(* IEC 61131-3 sources: ecmc_strucpp_app_example/st, 7 files *)

(* ---- el7041_velocity.st ---- *)
PROGRAM EL7041_VELOCITY
VAR
  actual_position    AT %IW0 : INT;   // @ecmc ec0.s14.positionActual01
  drive_control      AT %QW0 : WORD;  // @ecmc ec0.s14.driveControl01
  velocity_setpoint  AT %QW2 : INT;   // @ecmc ec0.s14.velocitySetpoint01
END_VAR

drive_control := 16#0001;
velocity_setpoint := 1000;
END_PROGRAM

(* ---- machine.st ---- *)
PROGRAM MACHINE
VAR
  start_button   AT %IX0.0 : BOOL;  // @ecmc ec0.s2.mm.inputDataArray01
  stop_button    AT %IX0.1 : BOOL;  // @ecmc ec0.s2.mm.inputDataArray01
  enable_output  AT %QX0.0 : BOOL;  // @ecmc ec0.s2.mm.outputDataArray01
  target_word    AT %QW2   : INT;   // @ecmc ec0.s2.mm.outputDataArray01
  counter        AT %MW0   : INT;
END_VAR

IF stop_button THEN
  enable_output := FALSE;
ELSIF start_button THEN
  enable_output := TRUE;
END_IF;

IF enable_output THEN
  counter := counter + 1;
  target_word := counter;
ELSE
  target_word := 0;
END_IF;
END_PROGRAM

(* ---- mc_power_move_absolute_lib.st ---- *)
PROGRAM MC_POWER_MOVE_ABSOLUTE_LIB
VAR
  axis        : ECMC_AXIS_REF;
  power       : MC_Power;
  moveAbs     : MC_MoveAbsolute;
  readPos     : MC_ReadActualPosition;

  enableCmd   AT %IX0.0 : BOOL;
  executeCmd  AT %IX0.1 : BOOL;

  targetPos   AT %IL8  : LREAL;
  velocity    AT %IL16 : LREAL;
  accel       AT %IL24 : LREAL;
  decel       AT %IL32 : LREAL;

  powerStatus AT %QX0.0 : BOOL;
  powerValid  AT %QX0.1 : BOOL;
  moveBusy    AT %QX0.2 : BOOL;
  moveDone    AT %QX0.3 : BOOL;
  moveError   AT %QX0.4 : BOOL;
  moveErrorId AT %QD4   : UDINT;
  actualPos   AT %QL8   : LREAL;
END_VAR

axis.AxisIndex := 0;

power(Axis := axis, Enable := enableCmd);
moveAbs(Axis := axis,
        Execute := executeCmd,
        Position := targetPos,
        Velocity := velocity,
        Acceleration := accel,
        Deceleration := decel);
readPos(Axis := axis, Enable := TRUE);

powerStatus := power.Status;
powerValid  := power.Valid;
moveBusy    := moveAbs.Busy;
moveDone    := moveAbs.Done;
moveError   := moveAbs.Error;
moveErrorId := moveAbs.ErrorID;
actualPos   := readPos.Position;
END_PROGRAM

(* ---- mc_power_move_relative_lib.st ---- *)
PROGRAM MC_POWER_MOVE_RELATIVE_LIB
VAR
  axis         : ECMC_AXIS_REF;
  power        : MC_Power;
  moveRel      : MC_MoveRelative;
  readStatus   : MC_ReadStatus;
  readPos      : MC_ReadActualPosition;

  enableCmd    AT %IX0.0 : BOOL;
  executeCmd   AT %IX0.1 : BOOL;

  distanceCmd  AT %IL8  : LREAL;
  velocityCmd  AT %IL16 : LREAL;
  accelCmd     AT %IL24 : LREAL;
  decelCmd     AT %IL32 : LREAL;

  powerStatus  AT %QX0.0 : BOOL;
  powerValid   AT %QX0.1 : BOOL;
  moveBusy     AT %QX0.2 : BOOL;
  moveDone     AT %QX0.3 : BOOL;
  moveError    AT %QX0.4 : BOOL;
  standStill   AT %QX0.5 : BOOL;
  discreteMove AT %QX0.6 : BOOL;
  errorStop    AT %QX0.7 : BOOL;
  moveErrorId  AT %QD4   : UDINT;
  actualPos    AT %QL8   : LREAL;
END_VAR

axis.AxisIndex := 0;

power(Axis := axis, Enable := enableCmd);
moveRel(Axis := axis,
        Execute := executeCmd,
        Distance := distanceCmd,
        Velocity := velocityCmd,
        Acceleration := accelCmd,
        Deceleration := decelCmd);
readStatus(Axis := axis, Enable := TRUE);
readPos(Axis := axis, Enable := TRUE);

powerStatus  := power.Status;
powerValid   := power.Valid;
moveBusy     := moveRel.Busy;
moveDone     := moveRel.Done;
moveError    := moveRel.Error;
standStill   := readStatus.StandStill;
discreteMove := readStatus.DiscreteMotion;
errorStop    := readStatus.ErrorStop;
moveErrorId  := moveRel.ErrorID;
actualPos    := readPos.Position;
END_PROGRAM

(* ---- mc_power_move_velocity_lib.st ---- *)
PROGRAM MC_POWER_MOVE_VELOCITY_LIB
VAR
  axis        : ECMC_AXIS_REF;
  power       : MC_Power;
  moveVel     : MC_MoveVelocity;
  readStatus  : MC_ReadStatus;
  readVel     : MC_ReadActualVelocity;

  enableCmd   AT %IX0.0 : BOOL;
  executeCmd  AT %IX0.1 : BOOL;

  velocityCmd AT %IL8  : LREAL;
  accelCmd    AT %IL16 : LREAL;
  decelCmd    AT %IL24 : LREAL;

  powerStatus AT %QX0.0 : BOOL;
  powerValid  AT %QX0.1 : BOOL;
  inVelocity  AT %QX0.2 : BOOL;
  moveBusy    AT %QX0.3 : BOOL;
  moveError   AT %QX0.4 : BOOL;
  standStill  AT %QX0.5 : BOOL;
  contMotion  AT %QX0.6 : BOOL;
  errorStop   AT %QX0.7 : BOOL;
  moveErrorId AT %QD4   : UDINT;
  actualVel   AT %QL8   : LREAL;
END_VAR

axis.AxisIndex := 0;

power(Axis := axis, Enable := enableCmd);
moveVel(Axis := axis,
        Execute := executeCmd,
        Velocity := velocityCmd,
        Acceleration := accelCmd,
        Deceleration := decelCmd);
readStatus(Axis := axis, Enable := TRUE);
readVel(Axis := axis, Enable := TRUE);

powerStatus := power.Status;
powerValid  := power.Valid;
inVelocity  := moveVel.InVelocity;
moveBusy    := moveVel.Busy;
moveError   := moveVel.Error;
standStill  := readStatus.StandStill;
contMotion  := readStatus.ContinuousMotion;
errorStop   := readStatus.ErrorStop;
moveErrorId := moveVel.ErrorID;
actualVel   := readVel.Velocity;
END_PROGRAM

(* ---- motion_actpos_mirror.st ---- *)
PROGRAM MOTION_ACTPOS_MIRROR
VAR
  source_actpos   AT %IL0 : LREAL;  // @ecmc ax1.enc.actpos
  target_position AT %QL0 : LREAL;  // @ecmc ax1.traj.targetpos
END_VAR

target_position := source_actpos;
END_PROGRAM

(* ---- motion_velocity_direct.st ---- *)
PROGRAM MOTION_VELOCITY_DIRECT
VAR
  actual_position  AT %IL0   : LREAL;  // @ecmc ax1.enc.actpos
  target_velocity  AT %QL0   : LREAL;  // @ecmc ax1.traj.targetvel
  drive_enable     AT %QX8.0 : BOOL;   // @ecmc ax1.drv.enable
END_VAR

drive_enable := TRUE;

IF actual_position < 1000.0 THEN
  target_velocity := 10.0;
ELSE
  target_velocity := -10.0;
END_IF;
END_PROGRAM
